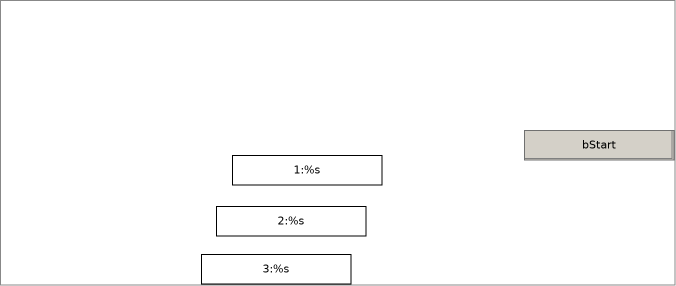
VISUALIZATION hmi  // 676x286
    Button (524,130 150x30), "bStart"
        toggle MAIN.bStart
    Rectangle (232,155 150x30), "1:%s", text variable: MAIN.strPara[1]
    Rectangle (216,206 150x30), "2:%s", text variable: MAIN.strPara[2]
    Rectangle (201,254 150x30), "3:%s", text variable: MAIN.strPara[3]
END_VISUALIZATION

(* stored: Version 1.1.0.1, ProductVersion 3.1.4022.12
   Visu hmi: Id {9b7d8372-a410-4fd8-bf29-a4ddacecd773} *)
